FUNCTION ARR_MAX (* Array Maximum *)
  (* Standard: 61499-1 *)
  (* Version 1.0, 2026-01-23, Franz Höpfinger, Andreas Demmler Fahrzeugbau, inspired by MAX in IEC 61131 Paper *)
  PACKAGE logiBUS::utils::dyn_arr;
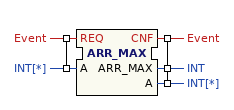
  EVENT_INPUT
    REQ WITH A;
  END_EVENT
  EVENT_OUTPUT
    CNF WITH ARR_MAX, A;
  END_EVENT
  VAR_OUTPUT
    ARR_MAX : INT;
  END_VAR
  VAR_IN_OUT
    A : ARRAY [*] OF INT; (* Input *)
  END_VAR
  BODY IN ST:
PACKAGE logiBUS::utils::dyn_arr;

(* Array Maximum *)
FUNCTION ARR_MAX : INT

VAR_IN_OUT
	A : ARRAY[*] OF INT; // Input
END_VAR

VAR_TEMP
	i : INT;
	currentMax : INT;
END_VAR

i := LOWER_BOUND(A, 1);
currentMax := A[i];
FOR i := LOWER_BOUND(A,1) + 1 TO UPPER_BOUND(A,1) DO
	currentMax := MAX(A[i], currentMax);

END_FOR;
ARR_MAX := currentMax;

END_FUNCTION
  END_BODY
END_FUNCTION
